INTERFACE ITFManual

END_INTERFACE

(* stored: Version 1.1.0.1, ProductVersion 3.1.4022.10
   Itf ITFManual: Id {3843b094-c537-4e85-aef2-142734ae0685} *)
